Fanuc KAREL source: kx00024.KL

-- PROVISIONAL review KL for V940-1; original PC SHA256 0bf744d95aab928c04adff277a5e637e283f93bad55d1834739da72a4a3449cc
-- Incomplete behavior may be omitted. Consult companion uncertainty JSON. Do not deploy.
PROGRAM KX00024
%NOLOCKGROUP
VAR
  I : INTEGER
  J : INTEGER
  B : BOOLEAN
  F : FILE
  S : STRING[80]
-- UNRESOLVED_DECL P type=000102
-- UNRESOLVED_DECL CNF type=00001c
BEGIN
  -- V9_ZERO_TABLE_METADATA_HINT layout=0001; no indexed target words; source/name/runtime held
  -- UNRESOLVED_PC offsets 5-15; opcodes 9D,22,A5
  -- UNRESOLVED_PC offsets 20-35; opcodes 22,A4,23
  -- UNRESOLVED_PC offsets 40-44; opcodes 7F
END KX00024
